INTERFACE I_MutCompList EXTENDS I_CompList

METHOD Append : Result
VAR_INPUT
	iComponent	: I_Component;
	nIndex		: UDINT;
END_VAR
END_METHOD

END_INTERFACE

(* stored: Version 1.1.0.1
   Itf I_MutCompList: Id {c2d0d42a-2de4-4c5c-b38b-df90732b2bb6}
   Method Append: Id {5c77e0e9-4c2a-4778-92ac-45cbb94f65af} *)
